ADAPTER IResetValves (* Adapter Interface *)
  (* Standard: 61499-1 *)
  (* Version 0.0, 7/6/2026, Schneider Electric *)
  PACKAGE SE.Nereda;
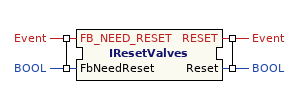
  EVENT_INPUT
    FB_NEED_RESET WITH FbNeedReset;
  END_EVENT
  EVENT_OUTPUT
    RESET WITH Reset;
  END_EVENT
  VAR_INPUT
    FbNeedReset : BOOL;
  END_VAR
  VAR_OUTPUT
    Reset : BOOL;
  END_VAR
  SERVICE SOCKET/PLUG
    SEQUENCE request_confirm
      SOCKET.REQ(REQD) -> PLUG.REQ(REQD);
      PLUG.CNF(CNFD) -> SOCKET.CNF(CNFD);
    END_SEQUENCE
    SEQUENCE indication_response
      PLUG.IND(INDD) -> SOCKET.IND(INDD);
      SOCKET.RSP(RSPD) -> PLUG.RSP(RSPD);
    END_SEQUENCE
  END_SERVICE
END_ADAPTER
